{attribute 'GeneratedUsingTerminal: ELX5151-0000-0016'}
{attribute addProperty BoxType "ELX5151-0000-0016"}
{attribute addProperty Id "Set_counterBOOL1"}
{attribute addProperty CRC "3181003151"}
{attribute addProperty Size "1"}
TYPE Control_BD9A418F :
STRUCT
	{attribute addProperty Name "Set_counter"}
	Set_counter : BOOL;
END_STRUCT
END_TYPE

(* stored: Version 1.2.0.0, ProductVersion 3.1.4024.9
   DUT Control_BD9A418F: Id {c5e59ca5-9723-48d4-82f0-14a9c9e89b98} *)
